(* IEC 61131-3 sources: repolevel_ST_code_completion/real_groud_truth最新/repoeval_elevator/full_result, 5 files *)

(* ---- F_DetectCurrentFloor.st ---- *)
FUNCTION F_DetectCurrentFloor : INT
VAR_INPUT
	FloorSensor0	:	BOOL;		// 0楼传感器
	FloorSensor1	:	BOOL;		// 1楼传感器
	FloorSensor2	:	BOOL;		// 2楼传感器
	FloorSensor3	:	BOOL;		// 3楼传感器
	CurrentFloor	:	INT;		// 当前楼层（用于保持状态）
END_VAR

VAR_OUTPUT
	DetectedFloor	:	INT;		// 检测到的楼层
END_VAR

// 检测当前楼层
IF FloorSensor0 THEN
	DetectedFloor := 0;
ELSIF FloorSensor1 THEN
	DetectedFloor := 1;
ELSIF FloorSensor2 THEN
	DetectedFloor := 2;
ELSIF FloorSensor3 THEN
	DetectedFloor := 3;
ELSE
	DetectedFloor := CurrentFloor; // 如果没有传感器触发，保持当前楼层
END_IF

RETURN DetectedFloor;
END_FUNCTION

// --------------------------------------------------
// Continue PLC_PRG logic
// --------------------------------------------------

// 更新当前楼层
CurrentFloor := F_DetectCurrentFloor(
	FloorSensor0 := FloorSensor0,
	FloorSensor1 := FloorSensor1,
	FloorSensor2 := FloorSensor2,
	FloorSensor3 := FloorSensor3,
	CurrentFloor := CurrentFloor
);

// ========== 呼叫处理 ==========
F_RegisterCalls(
	CallGround := CallGround,
	CallFloor1 := CallFloor1,
	CallFloor2 := CallFloor2,
	CallFloor3 := CallFloor3,
	TargetFloors := TargetFloors
);

// ========== 门控制逻辑 ==========
fbDoorController(
	bArrivedAtTarget := TargetFloors[CurrentFloor],
	bDoorClosed := DoorClosed
);
OpenDoor := fbDoorController.OpenDoor;
CloseDoor := fbDoorController.CloseDoor;

// ========== 电梯移动逻辑 ==========
fbMovementController(
	CurrentFloor := CurrentFloor,
	bDoorReady := DoorClosed,
	TargetFloors := TargetFloors
);

// 动画更新
aniDoor0 := fbDoorController.aniDoor0;
aniDoor1 := fbDoorController.aniDoor1;
aniDoor2 := fbDoorController.aniDoor2;
aniDoor3 := fbDoorController.aniDoor3;

// END PROGRAM PLC_PRG
END_FUNCTION

(* ---- F_RegisterCalls.st ---- *)
FUNCTION F_RegisterCalls
VAR_INPUT
	CallGround		:	BOOL;		// 0楼呼叫
	CallFloor1		:	BOOL;		// 1楼呼叫
	CallFloor2		:	BOOL;		// 2楼呼叫
	CallFloor3		:	BOOL;		// 3楼呼叫
END_VAR
VAR_IN_OUT
	TargetFloors	:	ARRAY[0..3] OF BOOL;	// 目标楼层数组
END_VAR

VAR
	i				:	INT;		// 循环变量
END_VAR

// 将呼叫信号注册到目标楼层数组中
IF CallGround THEN
	TargetFloors[0] := TRUE;
END_IF;

IF CallFloor1 THEN
	TargetFloors[1] := TRUE;
END_IF;

IF CallFloor2 THEN
	TargetFloors[2] := TRUE;
END_IF;

IF CallFloor3 THEN
	TargetFloors[3] := TRUE;
END_IF;

// 确保目标楼层数组的状态正确
FOR i := 0 TO 3 DO
	IF TargetFloors[i] THEN
		// 目标楼层已被注册
		// 可在此处添加调试或日志记录代码
	END_IF;
END_FOR;
END_FUNCTION

(* ---- F_UpdateDoorAnimation.st ---- *)
FUNCTION F_UpdateDoorAnimation : DINT
VAR_INPUT
	bOpenDoor		:	BOOL;		// 开门命令
	bCloseDoor		:	BOOL;		// 关门命令
	bCallFloor		:	BOOL;		// 该楼层有呼叫
	nCurrentAni		:	DINT;		// 当前动画值
	nMaxAni			:	DINT := 70;	// 最大动画值
END_VAR

VAR_OUTPUT
	nUpdatedAni		:	DINT;		// 更新后的动画值
END_VAR
VAR
	nStep			:	DINT := 5;	// 动画步长
END_VAR

// 检查是否需要开门动画
IF bOpenDoor THEN
	IF nCurrentAni < nMaxAni THEN
		nUpdatedAni := nCurrentAni + nStep; // 增加动画值
	ELSE
		nUpdatedAni := nMaxAni; // 达到最大动画值
	END_IF;
ELSIF bCloseDoor THEN
	IF nCurrentAni > 0 THEN
		nUpdatedAni := nCurrentAni - nStep; // 减少动画值
	ELSE
		nUpdatedAni := 0; // 达到最小动画值
	END_IF;
ELSE
	// 如果没有开门或关门命令，保持当前动画值
	nUpdatedAni := nCurrentAni;
END_IF;

// 返回更新后的动画值
RETURN nUpdatedAni;
END_FUNCTION

(* ---- FB_ElevatorDoorController.st ---- *)
FUNCTION_BLOCK FB_ElevatorDoorController
VAR_INPUT
	bArrivedAtTarget	:	BOOL;		// 到达目标楼层
	bDoorClosed			:	BOOL;		// 门已关闭传感器
END_VAR
VAR_OUTPUT
	bOpenDoor			:	BOOL;		// 开门命令
	bCloseDoor			:	BOOL;		// 关门命令
	bDoorOpen			:	BOOL;		// 门打开状态
	bDoorReady			:	BOOL;		// 门准备好（可以移动）
END_VAR

VAR
	fbDoorTimer			:	TON;		// 门操作定时器
	bDoorOpening		:	BOOL;		// 门正在打开
	bDoorClosing		:	BOOL;		// 门正在关闭
END_VAR

// 门控制逻辑
IF bArrivedAtTarget THEN
	// 如果到达目标楼层，且门未打开，则发送开门命令
	IF NOT bDoorOpen THEN
		bOpenDoor := TRUE;
		bCloseDoor := FALSE;
		bDoorOpening := TRUE;
		bDoorClosing := FALSE;
		fbDoorTimer(IN := TRUE, PT := T#5S); // 开门延时
	END_IF
ELSE
	// 如果未到达目标楼层，且门已打开，则发送关门命令
	IF bDoorOpen THEN
		bOpenDoor := FALSE;
		bCloseDoor := TRUE;
		bDoorOpening := FALSE;
		bDoorClosing := TRUE;
		fbDoorTimer(IN := TRUE, PT := T#5S); // 关门延时
	END_IF
END_IF

// 定时器完成后更新门状态
IF fbDoorTimer.Q THEN
	IF bDoorOpening THEN
		bDoorOpen := TRUE;
		bDoorReady := TRUE; // 门准备好，电梯可以移动
		bDoorOpening := FALSE;
	ELSEIF bDoorClosing THEN
		bDoorOpen := FALSE;
		bDoorReady := FALSE; // 门未准备好，电梯不能移动
		bDoorClosing := FALSE;
	END_IF
	fbDoorTimer(IN := FALSE); // 停止定时器
END_IF
END_FUNCTION_BLOCK

(* ---- FB_ElevatorMovement.st ---- *)
FUNCTION_BLOCK FB_ElevatorMovement
VAR_INPUT
	CurrentFloor		:	INT;				// 当前楼层
	bDoorReady			:	BOOL;				// 门准备好
END_VAR
VAR_IN_OUT
	TargetFloors		:	ARRAY[0..3] OF BOOL;	// 目标楼层数组
END_VAR
VAR_OUTPUT
	bMovingUp			:	BOOL;				// 向上移动
	bMovingDown			:	BOOL;				// 向下移动
	bArrivedAtTarget	:	BOOL;				// 到达目标楼层
END_VAR

VAR
	nTargetFloor		:	INT;				// 当前目标楼层
	nState				:	INT;				// 状态机
END_VAR

CASE nState OF
	0: // 空闲状态
		bMovingUp := FALSE;
		bMovingDown := FALSE;
		bArrivedAtTarget := FALSE;

		// 检查是否有目标楼层
		FOR i := 0 TO 3 DO
			IF TargetFloors[i] THEN
				nTargetFloor := i;
				nState := 1; // 开始移动流程
				EXIT;
			END_IF
		END_FOR

	1: // 移动到目标楼层
		IF CurrentFloor < nTargetFloor THEN
			bMovingUp := TRUE;
			bMovingDown := FALSE;
		ELSIF CurrentFloor > nTargetFloor THEN
			bMovingUp := FALSE;
			bMovingDown := TRUE;
		ELSE
			bMovingUp := FALSE;
			bMovingDown := FALSE;
			bArrivedAtTarget := TRUE;
			TargetFloors[nTargetFloor] := FALSE; // 清除目标楼层
			nState := 2; // 到达目标楼层
		END_IF

	2: // 等待门准备好
		IF bDoorReady THEN
			nState := 0; // 返回空闲状态
		END_IF
END_CASE
END_FUNCTION_BLOCK
